TYPE ST_PROCESS_DATA :
STRUCT
  nProcessId          : e_instance; // target process
  {attribute 'displaymode':='bin'}
  wTarget             : T_PROCESS;  // where and how many stations are to be used in process
END_STRUCT
END_TYPE

(* stored: Version 1.1.0.1, ProductVersion 3.1.4026.18
   DUT ST_PROCESS_DATA: Id {10da316b-4afc-4833-b500-703877710b1e} *)
